// TIA Portal V16 export
// export: Created 2023-03-29T11:03:21.8786625Z, ExportSetting WithDefaults, DisplayName Totally Integrated Automation Portal, DisplayVersion V16 Update 6, DisplayName TIA Portal Version Control Interface, DisplayVersion V16 Update 2, DisplayName TIA Portal Openness, DisplayVersion V16 Update 6, DisplayName STEP 7 Professional, DisplayVersion V16 Update 6, DisplayName STEP 7 Safety, DisplayVersion V16, DisplayName WinCC Advanced, DisplayVersion V16 Update 6
FUNCTION "Gotowość_i_Sygnalizacja" : Void   // FC8, LAD
TITLE = Ustawienie Gotowośći
{ S7_Optimized_Access := 'TRUE' }
AUTHOR : rtecmer
VERSION : 0.1
// Funkcja w zależności od przełącznika technologiczne związanego z przebudową zasuw z Czeskich na AUMA przełącza sygnał godowości w zależności jak ajest zasuwa podłączona w procesie technologicznym
// stored: AutoNumber true, IsIECCheckEnabled false, SetENOAutomatically false, UDAEnableTagReadback false
   VAR_TEMP   // added for the SCL form of the ladder/FBD networks
      _w1 : Bool;
   END_VAR
BEGIN

REGION Network 1 (SCL): Pływaki minimum - Zbiorniki Zb1 - 4
   // min pływak
   "Zmienne_sterujące_zbiorników".Zbiornik_1.is_min_float_Zb := "float_min_tank_1";
   "Zmienne_sterujące_zbiorników".Zbiornik_2.is_min_float_Zb := "float_min_tank_2";
   "Zmienne_sterujące_zbiorników".Zbiornik_3.is_min_float_Zb := "float_min_tank_3";
   "Zmienne_sterujące_zbiorników".Zbiornik_4.is_min_float_Zb := "float_min_tank_4";
   // max pływak
   "Zmienne_sterujące_zbiorników".Zbiornik_1.is_max_float_Zb := "float_max_tank_1";
   "Zmienne_sterujące_zbiorników".Zbiornik_2.is_max_float_Zb := "float_max_tank_2";
   "Zmienne_sterujące_zbiorników".Zbiornik_3.is_max_float_Zb := "float_max_tank_3";
   "Zmienne_sterujące_zbiorników".Zbiornik_4.is_max_float_Zb := "float_max_tank_4";
END_REGION

REGION Network 2: bit gotowości wspólny Z10
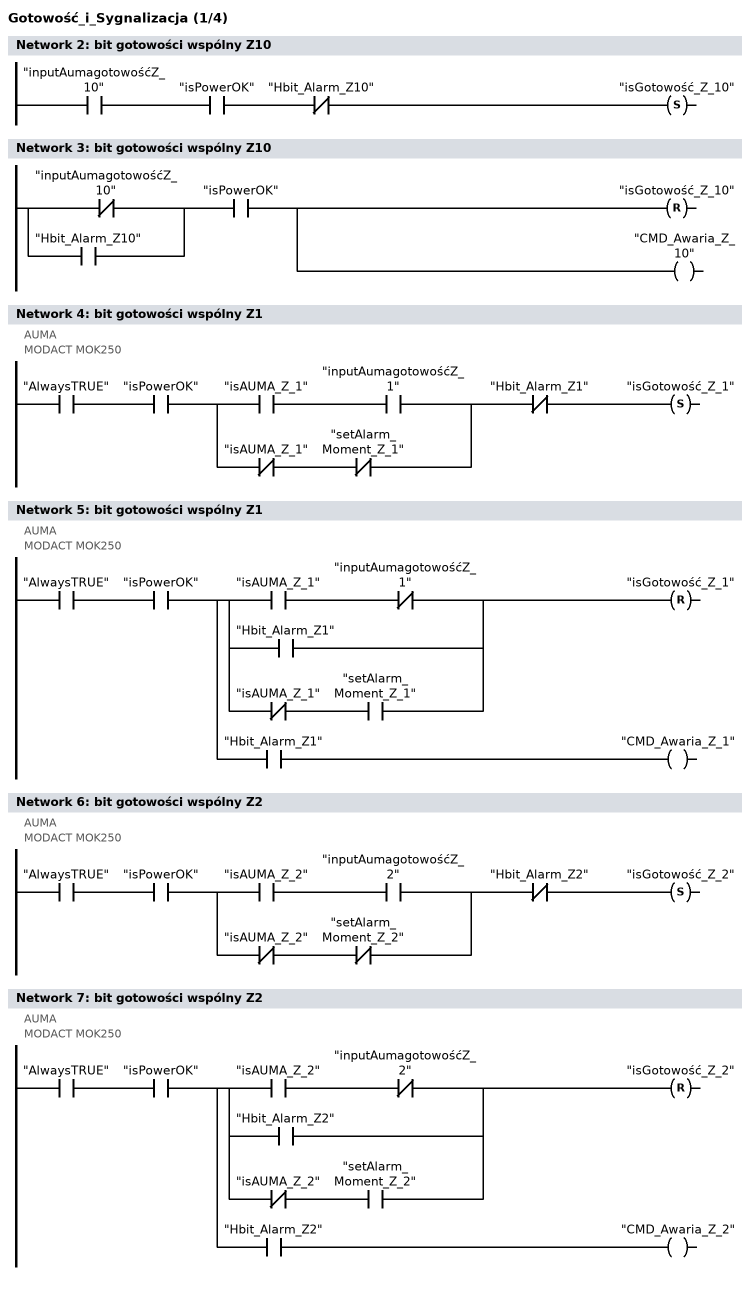
   RUNG wire#powerrail
      Contact( "inputAumagotowośćZ_10" )
      Contact( "isPowerOK" )
      I_Contact( "Hbit_Alarm_Z10" )
      S_Coil( "isGotowość_Z_10" )
   END_RUNG
   // the same network as SCL:
   IF "inputAumagotowośćZ_10" AND "isPowerOK" AND NOT "Hbit_Alarm_Z10" THEN
       "isGotowość_Z_10" := TRUE;
   END_IF;
END_REGION

REGION Network 3: bit gotowości wspólny Z10
   RUNG wire#powerrail
      I_Contact( "inputAumagotowośćZ_10" )
      wire#w1
      Contact( "isPowerOK" )
      wire#w2
      R_Coil( "isGotowość_Z_10" )
   END_RUNG
   RUNG wire#powerrail
      Contact( "Hbit_Alarm_Z10" )
   END_RUNG wire#w1
   RUNG wire#w2
      Coil( "CMD_Awaria_Z_10" )
   END_RUNG
   // the same network as SCL:
   #_w1 := (NOT "inputAumagotowośćZ_10" OR "Hbit_Alarm_Z10") AND "isPowerOK";
   IF #_w1 THEN "isGotowość_Z_10" := FALSE; END_IF;
   "CMD_Awaria_Z_10" := #_w1;
END_REGION

REGION Network 4: bit gotowości wspólny Z1
   // AUMA
   // MODACT MOK250
   RUNG wire#powerrail
      Contact( "AlwaysTRUE" )
      Contact( "isPowerOK" )
      wire#w1
      Contact( "isAUMA_Z_1" )
      Contact( "inputAumagotowośćZ_1" )
      wire#w2
      I_Contact( "Hbit_Alarm_Z1" )
      S_Coil( "isGotowość_Z_1" )
   END_RUNG
   RUNG wire#w1
      I_Contact( "isAUMA_Z_1" )
      I_Contact( "setAlarm_Moment_Z_1" )
   END_RUNG wire#w2
   // the same network as SCL:
   IF "AlwaysTRUE" AND "isPowerOK" AND (("isAUMA_Z_1" AND "inputAumagotowośćZ_1") OR (NOT "isAUMA_Z_1" AND NOT "setAlarm_Moment_Z_1")) AND NOT "Hbit_Alarm_Z1" THEN
       "isGotowość_Z_1" := TRUE;
   END_IF;
END_REGION

REGION Network 5: bit gotowości wspólny Z1
   // AUMA
   // MODACT MOK250
   RUNG wire#powerrail
      Contact( "AlwaysTRUE" )
      Contact( "isPowerOK" )
      wire#w1
      Contact( "isAUMA_Z_1" )
      I_Contact( "inputAumagotowośćZ_1" )
      wire#w2
      R_Coil( "isGotowość_Z_1" )
   END_RUNG
   RUNG wire#w1
      Contact( "Hbit_Alarm_Z1" )
   END_RUNG wire#w2
   RUNG wire#w1
      I_Contact( "isAUMA_Z_1" )
      Contact( "setAlarm_Moment_Z_1" )
   END_RUNG wire#w2
   RUNG wire#w1
      Contact( "Hbit_Alarm_Z1" )
      Coil( "CMD_Awaria_Z_1" )
   END_RUNG
   // the same network as SCL:
   #_w1 := "AlwaysTRUE" AND "isPowerOK";
   IF #_w1 AND (("isAUMA_Z_1" AND NOT "inputAumagotowośćZ_1") OR "Hbit_Alarm_Z1" OR (NOT "isAUMA_Z_1" AND "setAlarm_Moment_Z_1")) THEN
       "isGotowość_Z_1" := FALSE;
   END_IF;
   "CMD_Awaria_Z_1" := #_w1 AND "Hbit_Alarm_Z1";
END_REGION

REGION Network 6: bit gotowości wspólny Z2
   // AUMA
   // MODACT MOK250
   RUNG wire#powerrail
      Contact( "AlwaysTRUE" )
      Contact( "isPowerOK" )
      wire#w1
      Contact( "isAUMA_Z_2" )
      Contact( "inputAumagotowośćZ_2" )
      wire#w2
      I_Contact( "Hbit_Alarm_Z2" )
      S_Coil( "isGotowość_Z_2" )
   END_RUNG
   RUNG wire#w1
      I_Contact( "isAUMA_Z_2" )
      I_Contact( "setAlarm_Moment_Z_2" )
   END_RUNG wire#w2
   // the same network as SCL:
   IF "AlwaysTRUE" AND "isPowerOK" AND (("isAUMA_Z_2" AND "inputAumagotowośćZ_2") OR (NOT "isAUMA_Z_2" AND NOT "setAlarm_Moment_Z_2")) AND NOT "Hbit_Alarm_Z2" THEN
       "isGotowość_Z_2" := TRUE;
   END_IF;
END_REGION

REGION Network 7: bit gotowości wspólny Z2
   // AUMA
   // MODACT MOK250
   RUNG wire#powerrail
      Contact( "AlwaysTRUE" )
      Contact( "isPowerOK" )
      wire#w1
      Contact( "isAUMA_Z_2" )
      I_Contact( "inputAumagotowośćZ_2" )
      wire#w2
      R_Coil( "isGotowość_Z_2" )
   END_RUNG
   RUNG wire#w1
      Contact( "Hbit_Alarm_Z2" )
   END_RUNG wire#w2
   RUNG wire#w1
      I_Contact( "isAUMA_Z_2" )
      Contact( "setAlarm_Moment_Z_2" )
   END_RUNG wire#w2
   RUNG wire#w1
      Contact( "Hbit_Alarm_Z2" )
      Coil( "CMD_Awaria_Z_2" )
   END_RUNG
   // the same network as SCL:
   #_w1 := "AlwaysTRUE" AND "isPowerOK";
   IF #_w1 AND (("isAUMA_Z_2" AND NOT "inputAumagotowośćZ_2") OR "Hbit_Alarm_Z2" OR (NOT "isAUMA_Z_2" AND "setAlarm_Moment_Z_2")) THEN
       "isGotowość_Z_2" := FALSE;
   END_IF;
   "CMD_Awaria_Z_2" := #_w1 AND "Hbit_Alarm_Z2";
END_REGION

REGION Network 8: bit gotowości wspólny Z3
   // AUMA
   // MODACT MOK250
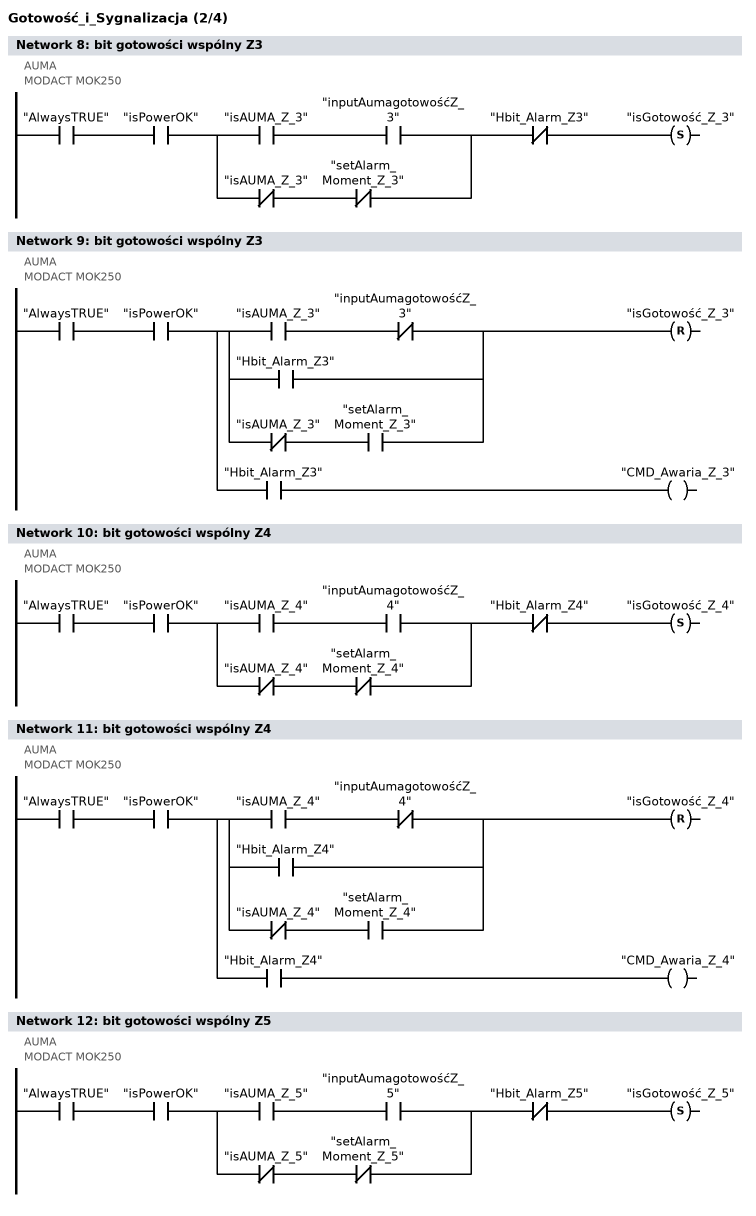
   RUNG wire#powerrail
      Contact( "AlwaysTRUE" )
      Contact( "isPowerOK" )
      wire#w1
      Contact( "isAUMA_Z_3" )
      Contact( "inputAumagotowośćZ_3" )
      wire#w2
      I_Contact( "Hbit_Alarm_Z3" )
      S_Coil( "isGotowość_Z_3" )
   END_RUNG
   RUNG wire#w1
      I_Contact( "isAUMA_Z_3" )
      I_Contact( "setAlarm_Moment_Z_3" )
   END_RUNG wire#w2
   // the same network as SCL:
   IF "AlwaysTRUE" AND "isPowerOK" AND (("isAUMA_Z_3" AND "inputAumagotowośćZ_3") OR (NOT "isAUMA_Z_3" AND NOT "setAlarm_Moment_Z_3")) AND NOT "Hbit_Alarm_Z3" THEN
       "isGotowość_Z_3" := TRUE;
   END_IF;
END_REGION

REGION Network 9: bit gotowości wspólny Z3
   // AUMA
   // MODACT MOK250
   RUNG wire#powerrail
      Contact( "AlwaysTRUE" )
      Contact( "isPowerOK" )
      wire#w1
      Contact( "isAUMA_Z_3" )
      I_Contact( "inputAumagotowośćZ_3" )
      wire#w2
      R_Coil( "isGotowość_Z_3" )
   END_RUNG
   RUNG wire#w1
      Contact( "Hbit_Alarm_Z3" )
   END_RUNG wire#w2
   RUNG wire#w1
      I_Contact( "isAUMA_Z_3" )
      Contact( "setAlarm_Moment_Z_3" )
   END_RUNG wire#w2
   RUNG wire#w1
      Contact( "Hbit_Alarm_Z3" )
      Coil( "CMD_Awaria_Z_3" )
   END_RUNG
   // the same network as SCL:
   #_w1 := "AlwaysTRUE" AND "isPowerOK";
   IF #_w1 AND (("isAUMA_Z_3" AND NOT "inputAumagotowośćZ_3") OR "Hbit_Alarm_Z3" OR (NOT "isAUMA_Z_3" AND "setAlarm_Moment_Z_3")) THEN
       "isGotowość_Z_3" := FALSE;
   END_IF;
   "CMD_Awaria_Z_3" := #_w1 AND "Hbit_Alarm_Z3";
END_REGION

REGION Network 10: bit gotowości wspólny Z4
   // AUMA
   // MODACT MOK250
   RUNG wire#powerrail
      Contact( "AlwaysTRUE" )
      Contact( "isPowerOK" )
      wire#w1
      Contact( "isAUMA_Z_4" )
      Contact( "inputAumagotowośćZ_4" )
      wire#w2
      I_Contact( "Hbit_Alarm_Z4" )
      S_Coil( "isGotowość_Z_4" )
   END_RUNG
   RUNG wire#w1
      I_Contact( "isAUMA_Z_4" )
      I_Contact( "setAlarm_Moment_Z_4" )
   END_RUNG wire#w2
   // the same network as SCL:
   IF "AlwaysTRUE" AND "isPowerOK" AND (("isAUMA_Z_4" AND "inputAumagotowośćZ_4") OR (NOT "isAUMA_Z_4" AND NOT "setAlarm_Moment_Z_4")) AND NOT "Hbit_Alarm_Z4" THEN
       "isGotowość_Z_4" := TRUE;
   END_IF;
END_REGION

REGION Network 11: bit gotowości wspólny Z4
   // AUMA
   // MODACT MOK250
   RUNG wire#powerrail
      Contact( "AlwaysTRUE" )
      Contact( "isPowerOK" )
      wire#w1
      Contact( "isAUMA_Z_4" )
      I_Contact( "inputAumagotowośćZ_4" )
      wire#w2
      R_Coil( "isGotowość_Z_4" )
   END_RUNG
   RUNG wire#w1
      Contact( "Hbit_Alarm_Z4" )
   END_RUNG wire#w2
   RUNG wire#w1
      I_Contact( "isAUMA_Z_4" )
      Contact( "setAlarm_Moment_Z_4" )
   END_RUNG wire#w2
   RUNG wire#w1
      Contact( "Hbit_Alarm_Z4" )
      Coil( "CMD_Awaria_Z_4" )
   END_RUNG
   // the same network as SCL:
   #_w1 := "AlwaysTRUE" AND "isPowerOK";
   IF #_w1 AND (("isAUMA_Z_4" AND NOT "inputAumagotowośćZ_4") OR "Hbit_Alarm_Z4" OR (NOT "isAUMA_Z_4" AND "setAlarm_Moment_Z_4")) THEN
       "isGotowość_Z_4" := FALSE;
   END_IF;
   "CMD_Awaria_Z_4" := #_w1 AND "Hbit_Alarm_Z4";
END_REGION

REGION Network 12: bit gotowości wspólny Z5
   // AUMA
   // MODACT MOK250
   RUNG wire#powerrail
      Contact( "AlwaysTRUE" )
      Contact( "isPowerOK" )
      wire#w1
      Contact( "isAUMA_Z_5" )
      Contact( "inputAumagotowośćZ_5" )
      wire#w2
      I_Contact( "Hbit_Alarm_Z5" )
      S_Coil( "isGotowość_Z_5" )
   END_RUNG
   RUNG wire#w1
      I_Contact( "isAUMA_Z_5" )
      I_Contact( "setAlarm_Moment_Z_5" )
   END_RUNG wire#w2
   // the same network as SCL:
   IF "AlwaysTRUE" AND "isPowerOK" AND (("isAUMA_Z_5" AND "inputAumagotowośćZ_5") OR (NOT "isAUMA_Z_5" AND NOT "setAlarm_Moment_Z_5")) AND NOT "Hbit_Alarm_Z5" THEN
       "isGotowość_Z_5" := TRUE;
   END_IF;
END_REGION

REGION Network 13: bit gotowości wspólny Z5
   // AUMA
   // MODACT MOK250
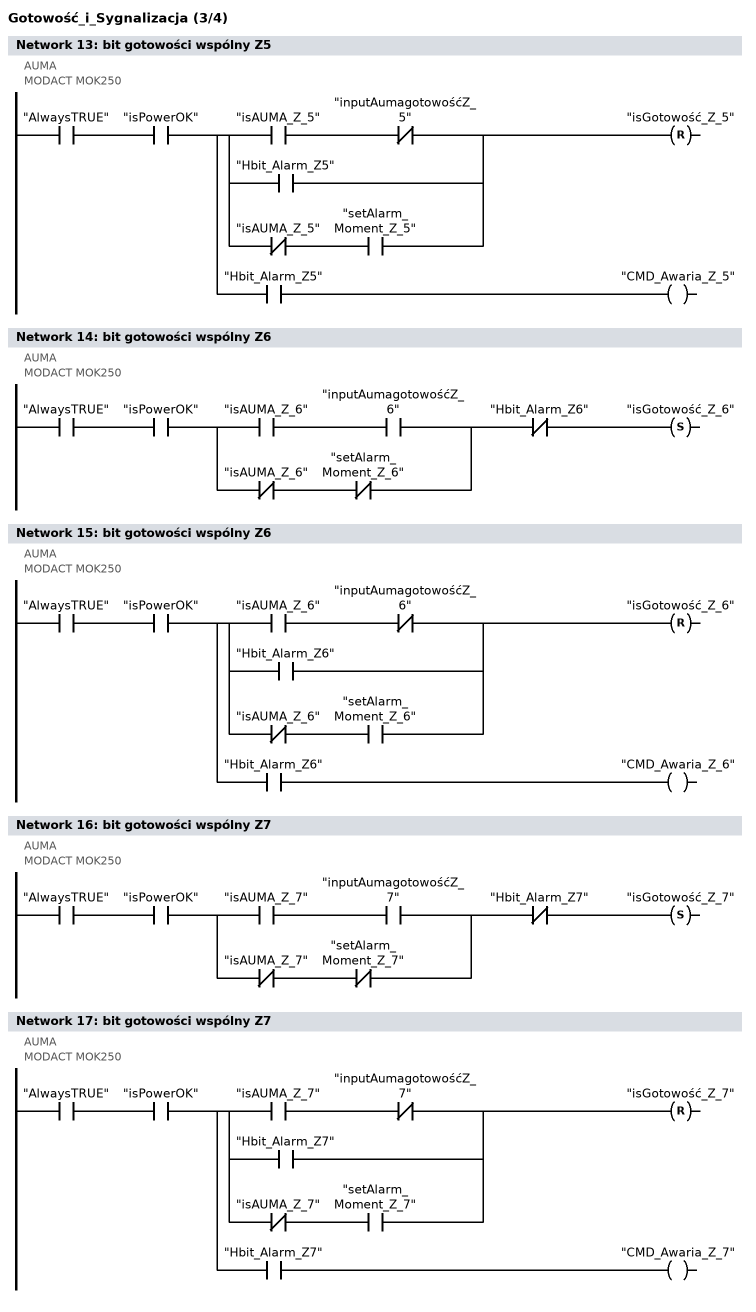
   RUNG wire#powerrail
      Contact( "AlwaysTRUE" )
      Contact( "isPowerOK" )
      wire#w1
      Contact( "isAUMA_Z_5" )
      I_Contact( "inputAumagotowośćZ_5" )
      wire#w2
      R_Coil( "isGotowość_Z_5" )
   END_RUNG
   RUNG wire#w1
      Contact( "Hbit_Alarm_Z5" )
   END_RUNG wire#w2
   RUNG wire#w1
      I_Contact( "isAUMA_Z_5" )
      Contact( "setAlarm_Moment_Z_5" )
   END_RUNG wire#w2
   RUNG wire#w1
      Contact( "Hbit_Alarm_Z5" )
      Coil( "CMD_Awaria_Z_5" )
   END_RUNG
   // the same network as SCL:
   #_w1 := "AlwaysTRUE" AND "isPowerOK";
   IF #_w1 AND (("isAUMA_Z_5" AND NOT "inputAumagotowośćZ_5") OR "Hbit_Alarm_Z5" OR (NOT "isAUMA_Z_5" AND "setAlarm_Moment_Z_5")) THEN
       "isGotowość_Z_5" := FALSE;
   END_IF;
   "CMD_Awaria_Z_5" := #_w1 AND "Hbit_Alarm_Z5";
END_REGION

REGION Network 14: bit gotowości wspólny Z6
   // AUMA
   // MODACT MOK250
   RUNG wire#powerrail
      Contact( "AlwaysTRUE" )
      Contact( "isPowerOK" )
      wire#w1
      Contact( "isAUMA_Z_6" )
      Contact( "inputAumagotowośćZ_6" )
      wire#w2
      I_Contact( "Hbit_Alarm_Z6" )
      S_Coil( "isGotowość_Z_6" )
   END_RUNG
   RUNG wire#w1
      I_Contact( "isAUMA_Z_6" )
      I_Contact( "setAlarm_Moment_Z_6" )
   END_RUNG wire#w2
   // the same network as SCL:
   IF "AlwaysTRUE" AND "isPowerOK" AND (("isAUMA_Z_6" AND "inputAumagotowośćZ_6") OR (NOT "isAUMA_Z_6" AND NOT "setAlarm_Moment_Z_6")) AND NOT "Hbit_Alarm_Z6" THEN
       "isGotowość_Z_6" := TRUE;
   END_IF;
END_REGION

REGION Network 15: bit gotowości wspólny Z6
   // AUMA
   // MODACT MOK250
   RUNG wire#powerrail
      Contact( "AlwaysTRUE" )
      Contact( "isPowerOK" )
      wire#w1
      Contact( "isAUMA_Z_6" )
      I_Contact( "inputAumagotowośćZ_6" )
      wire#w2
      R_Coil( "isGotowość_Z_6" )
   END_RUNG
   RUNG wire#w1
      Contact( "Hbit_Alarm_Z6" )
   END_RUNG wire#w2
   RUNG wire#w1
      I_Contact( "isAUMA_Z_6" )
      Contact( "setAlarm_Moment_Z_6" )
   END_RUNG wire#w2
   RUNG wire#w1
      Contact( "Hbit_Alarm_Z6" )
      Coil( "CMD_Awaria_Z_6" )
   END_RUNG
   // the same network as SCL:
   #_w1 := "AlwaysTRUE" AND "isPowerOK";
   IF #_w1 AND (("isAUMA_Z_6" AND NOT "inputAumagotowośćZ_6") OR "Hbit_Alarm_Z6" OR (NOT "isAUMA_Z_6" AND "setAlarm_Moment_Z_6")) THEN
       "isGotowość_Z_6" := FALSE;
   END_IF;
   "CMD_Awaria_Z_6" := #_w1 AND "Hbit_Alarm_Z6";
END_REGION

REGION Network 16: bit gotowości wspólny Z7
   // AUMA
   // MODACT MOK250
   RUNG wire#powerrail
      Contact( "AlwaysTRUE" )
      Contact( "isPowerOK" )
      wire#w1
      Contact( "isAUMA_Z_7" )
      Contact( "inputAumagotowośćZ_7" )
      wire#w2
      I_Contact( "Hbit_Alarm_Z7" )
      S_Coil( "isGotowość_Z_7" )
   END_RUNG
   RUNG wire#w1
      I_Contact( "isAUMA_Z_7" )
      I_Contact( "setAlarm_Moment_Z_7" )
   END_RUNG wire#w2
   // the same network as SCL:
   IF "AlwaysTRUE" AND "isPowerOK" AND (("isAUMA_Z_7" AND "inputAumagotowośćZ_7") OR (NOT "isAUMA_Z_7" AND NOT "setAlarm_Moment_Z_7")) AND NOT "Hbit_Alarm_Z7" THEN
       "isGotowość_Z_7" := TRUE;
   END_IF;
END_REGION

REGION Network 17: bit gotowości wspólny Z7
   // AUMA
   // MODACT MOK250
   RUNG wire#powerrail
      Contact( "AlwaysTRUE" )
      Contact( "isPowerOK" )
      wire#w1
      Contact( "isAUMA_Z_7" )
      I_Contact( "inputAumagotowośćZ_7" )
      wire#w2
      R_Coil( "isGotowość_Z_7" )
   END_RUNG
   RUNG wire#w1
      Contact( "Hbit_Alarm_Z7" )
   END_RUNG wire#w2
   RUNG wire#w1
      I_Contact( "isAUMA_Z_7" )
      Contact( "setAlarm_Moment_Z_7" )
   END_RUNG wire#w2
   RUNG wire#w1
      Contact( "Hbit_Alarm_Z7" )
      Coil( "CMD_Awaria_Z_7" )
   END_RUNG
   // the same network as SCL:
   #_w1 := "AlwaysTRUE" AND "isPowerOK";
   IF #_w1 AND (("isAUMA_Z_7" AND NOT "inputAumagotowośćZ_7") OR "Hbit_Alarm_Z7" OR (NOT "isAUMA_Z_7" AND "setAlarm_Moment_Z_7")) THEN
       "isGotowość_Z_7" := FALSE;
   END_IF;
   "CMD_Awaria_Z_7" := #_w1 AND "Hbit_Alarm_Z7";
END_REGION

REGION Network 18: bit gotowości wspólny Z8
   // AUMA
   // MODACT MOK250
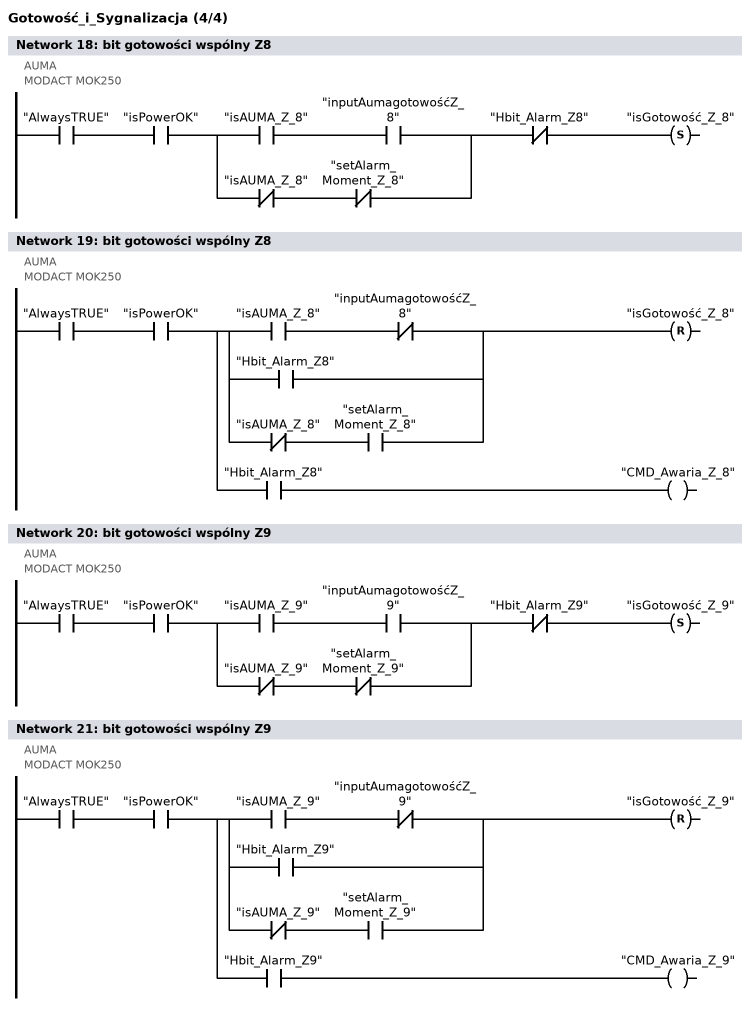
   RUNG wire#powerrail
      Contact( "AlwaysTRUE" )
      Contact( "isPowerOK" )
      wire#w1
      Contact( "isAUMA_Z_8" )
      Contact( "inputAumagotowośćZ_8" )
      wire#w2
      I_Contact( "Hbit_Alarm_Z8" )
      S_Coil( "isGotowość_Z_8" )
   END_RUNG
   RUNG wire#w1
      I_Contact( "isAUMA_Z_8" )
      I_Contact( "setAlarm_Moment_Z_8" )
   END_RUNG wire#w2
   // the same network as SCL:
   IF "AlwaysTRUE" AND "isPowerOK" AND (("isAUMA_Z_8" AND "inputAumagotowośćZ_8") OR (NOT "isAUMA_Z_8" AND NOT "setAlarm_Moment_Z_8")) AND NOT "Hbit_Alarm_Z8" THEN
       "isGotowość_Z_8" := TRUE;
   END_IF;
END_REGION

REGION Network 19: bit gotowości wspólny Z8
   // AUMA
   // MODACT MOK250
   RUNG wire#powerrail
      Contact( "AlwaysTRUE" )
      Contact( "isPowerOK" )
      wire#w1
      Contact( "isAUMA_Z_8" )
      I_Contact( "inputAumagotowośćZ_8" )
      wire#w2
      R_Coil( "isGotowość_Z_8" )
   END_RUNG
   RUNG wire#w1
      Contact( "Hbit_Alarm_Z8" )
   END_RUNG wire#w2
   RUNG wire#w1
      I_Contact( "isAUMA_Z_8" )
      Contact( "setAlarm_Moment_Z_8" )
   END_RUNG wire#w2
   RUNG wire#w1
      Contact( "Hbit_Alarm_Z8" )
      Coil( "CMD_Awaria_Z_8" )
   END_RUNG
   // the same network as SCL:
   #_w1 := "AlwaysTRUE" AND "isPowerOK";
   IF #_w1 AND (("isAUMA_Z_8" AND NOT "inputAumagotowośćZ_8") OR "Hbit_Alarm_Z8" OR (NOT "isAUMA_Z_8" AND "setAlarm_Moment_Z_8")) THEN
       "isGotowość_Z_8" := FALSE;
   END_IF;
   "CMD_Awaria_Z_8" := #_w1 AND "Hbit_Alarm_Z8";
END_REGION

REGION Network 20: bit gotowości wspólny Z9
   // AUMA
   // MODACT MOK250
   RUNG wire#powerrail
      Contact( "AlwaysTRUE" )
      Contact( "isPowerOK" )
      wire#w1
      Contact( "isAUMA_Z_9" )
      Contact( "inputAumagotowośćZ_9" )
      wire#w2
      I_Contact( "Hbit_Alarm_Z9" )
      S_Coil( "isGotowość_Z_9" )
   END_RUNG
   RUNG wire#w1
      I_Contact( "isAUMA_Z_9" )
      I_Contact( "setAlarm_Moment_Z_9" )
   END_RUNG wire#w2
   // the same network as SCL:
   IF "AlwaysTRUE" AND "isPowerOK" AND (("isAUMA_Z_9" AND "inputAumagotowośćZ_9") OR (NOT "isAUMA_Z_9" AND NOT "setAlarm_Moment_Z_9")) AND NOT "Hbit_Alarm_Z9" THEN
       "isGotowość_Z_9" := TRUE;
   END_IF;
END_REGION

REGION Network 21: bit gotowości wspólny Z9
   // AUMA
   // MODACT MOK250
   RUNG wire#powerrail
      Contact( "AlwaysTRUE" )
      Contact( "isPowerOK" )
      wire#w1
      Contact( "isAUMA_Z_9" )
      I_Contact( "inputAumagotowośćZ_9" )
      wire#w2
      R_Coil( "isGotowość_Z_9" )
   END_RUNG
   RUNG wire#w1
      Contact( "Hbit_Alarm_Z9" )
   END_RUNG wire#w2
   RUNG wire#w1
      I_Contact( "isAUMA_Z_9" )
      Contact( "setAlarm_Moment_Z_9" )
   END_RUNG wire#w2
   RUNG wire#w1
      Contact( "Hbit_Alarm_Z9" )
      Coil( "CMD_Awaria_Z_9" )
   END_RUNG
   // the same network as SCL:
   #_w1 := "AlwaysTRUE" AND "isPowerOK";
   IF #_w1 AND (("isAUMA_Z_9" AND NOT "inputAumagotowośćZ_9") OR "Hbit_Alarm_Z9" OR (NOT "isAUMA_Z_9" AND "setAlarm_Moment_Z_9")) THEN
       "isGotowość_Z_9" := FALSE;
   END_IF;
   "CMD_Awaria_Z_9" := #_w1 AND "Hbit_Alarm_Z9";
END_REGION
END_FUNCTION
